{attribute 'qualified_only'}
{attribute 'strict'}
TYPE stWorkStatus :
(
	None := 0,
	Started:=1,
	Completed:=2
)BYTE;
END_TYPE

(* stored: Version 1.1.0.1, ProductVersion 3.1.4024.9
   DUT stWorkStatus: Id {8fc868b1-c9ac-4df7-ada5-ef7f80145016} *)
